// TIA Portal V19 export
FUNCTION "CollectAlarms" : Void   // FC61, LAD
TITLE = Alarm Collector Unit
// Collects alarms from the respective level and categorises the alarms into the different alarm classes. Filling the alarm DB with specific alarm messages which are defined in the comment of the defined alarm. The definition of possible alarms within a equipment is handled here.
// stored: Namespace Unit2.EM2, SetENOAutomatically false
   VAR_INPUT
      resetAlarms : Bool;
      disableAlarms : Bool;
   END_VAR
   VAR_OUTPUT
      commandsToUnit : "LUC_typeStateCommands";   // Feedback to the unit
   END_VAR
BEGIN

REGION Network 1: Reset Alarms
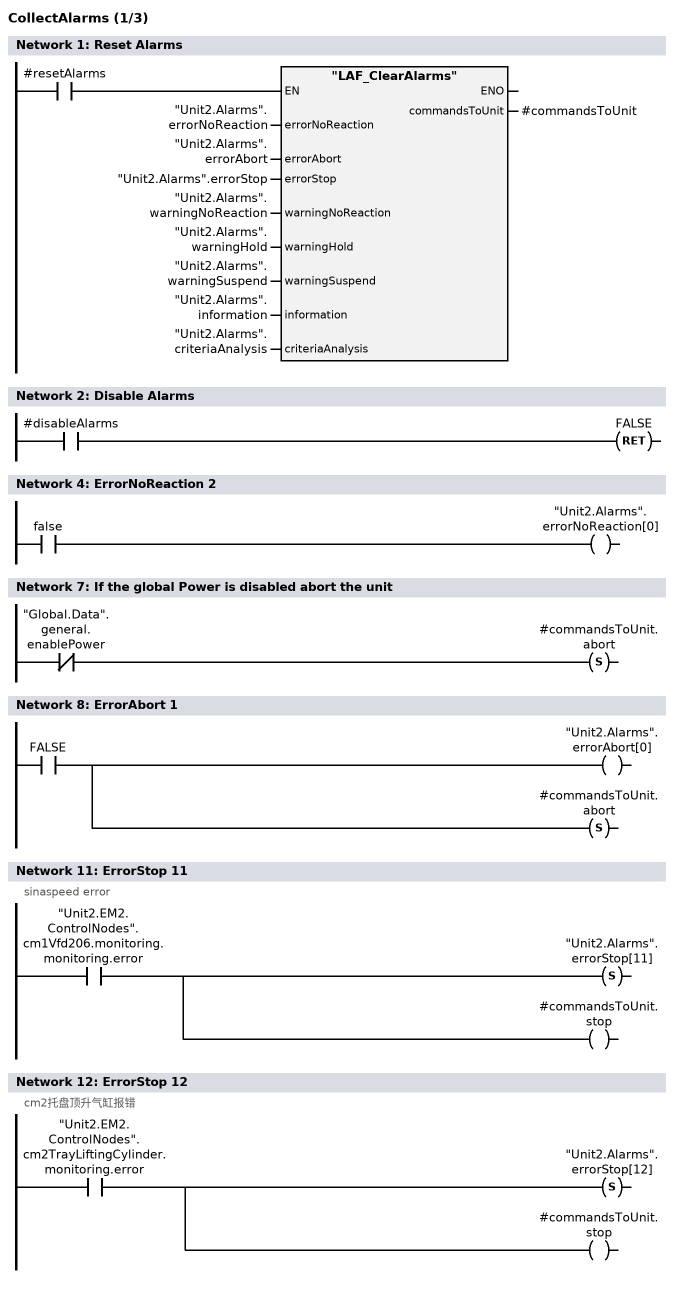
   RUNG wire#powerrail
      Contact( #resetAlarms )
      "LAF_ClearAlarms"(errorNoReaction := "Unit2.Alarms".errorNoReaction, errorAbort := "Unit2.Alarms".errorAbort, errorStop := "Unit2.Alarms".errorStop, warningNoReaction := "Unit2.Alarms".warningNoReaction, warningHold := "Unit2.Alarms".warningHold, warningSuspend := "Unit2.Alarms".warningSuspend, information := "Unit2.Alarms".information, criteriaAnalysis := "Unit2.Alarms".criteriaAnalysis, commandsToUnit => #commandsToUnit)
   END_RUNG
   // the same network as SCL:
   IF #resetAlarms THEN
       "LAF_ClearAlarms"(errorNoReaction := "Unit2.Alarms".errorNoReaction,
                         errorAbort := "Unit2.Alarms".errorAbort,
                         errorStop := "Unit2.Alarms".errorStop,
                         warningNoReaction := "Unit2.Alarms".warningNoReaction,
                         warningHold := "Unit2.Alarms".warningHold,
                         warningSuspend := "Unit2.Alarms".warningSuspend,
                         information := "Unit2.Alarms".information,
                         criteriaAnalysis := "Unit2.Alarms".criteriaAnalysis,
                         commandsToUnit => #commandsToUnit);
   END_IF;
END_REGION

REGION Network 2: Disable Alarms
   RUNG wire#powerrail
      Contact( #disableAlarms )
      ReturnCoil( FALSE )
   END_RUNG
   // the same network as SCL:
   IF #disableAlarms THEN
       ENO := FALSE;
       RETURN;
   END_IF;
END_REGION

REGION Network 3: *************** Error No Reaction ************************
END_REGION

REGION Network 4: ErrorNoReaction 2
   RUNG wire#powerrail
      Contact( false )
      Coil( "Unit2.Alarms".errorNoReaction[0] )
   END_RUNG
   // the same network as SCL:
   "Unit2.Alarms".errorNoReaction[0] := false;
END_REGION

REGION Network 6: *************** Error and Abort **************************
END_REGION

REGION Network 7: If the global Power is disabled abort the unit
   RUNG wire#powerrail
      I_Contact( "Global.Data".general.enablePower )
      S_Coil( #commandsToUnit.abort )
   END_RUNG
   // the same network as SCL:
   IF NOT "Global.Data".general.enablePower THEN #commandsToUnit.abort := TRUE; END_IF;
END_REGION

REGION Network 8: ErrorAbort 1
   RUNG wire#powerrail
      Contact( FALSE )
      wire#w1
      Coil( "Unit2.Alarms".errorAbort[0] )
   END_RUNG
   RUNG wire#w1
      S_Coil( #commandsToUnit.abort )
   END_RUNG
   // the same network as SCL:
   "Unit2.Alarms".errorAbort[0] := FALSE;
   IF FALSE THEN #commandsToUnit.abort := TRUE; END_IF;
END_REGION

REGION Network 10: *************** Error and Stop ***************************
END_REGION

REGION Network 11: ErrorStop 11
   // sinaspeed error
   RUNG wire#powerrail
      Contact( "Unit2.EM2.ControlNodes".cm1Vfd206.monitoring.monitoring.error )
      wire#w1
      S_Coil( "Unit2.Alarms".errorStop[11] )
   END_RUNG
   RUNG wire#w1
      Coil( #commandsToUnit.stop )
   END_RUNG
   // the same network as SCL:
   IF "Unit2.EM2.ControlNodes".cm1Vfd206.monitoring.monitoring.error THEN
       "Unit2.Alarms".errorStop[11] := TRUE;
   END_IF;
   #commandsToUnit.stop := "Unit2.EM2.ControlNodes".cm1Vfd206.monitoring.monitoring.error;
END_REGION

REGION Network 12: ErrorStop 12
   // cm2托盘顶升气缸报错
   RUNG wire#powerrail
      Contact( "Unit2.EM2.ControlNodes".cm2TrayLiftingCylinder.monitoring.error )
      wire#w1
      S_Coil( "Unit2.Alarms".errorStop[12] )
   END_RUNG
   RUNG wire#w1
      Coil( #commandsToUnit.stop )
   END_RUNG
   // the same network as SCL:
   IF "Unit2.EM2.ControlNodes".cm2TrayLiftingCylinder.monitoring.error THEN
       "Unit2.Alarms".errorStop[12] := TRUE;
   END_IF;
   #commandsToUnit.stop := "Unit2.EM2.ControlNodes".cm2TrayLiftingCylinder.monitoring.error;
END_REGION

REGION Network 13: ErrorStop 13
   // cm3电芯顶升气缸报错
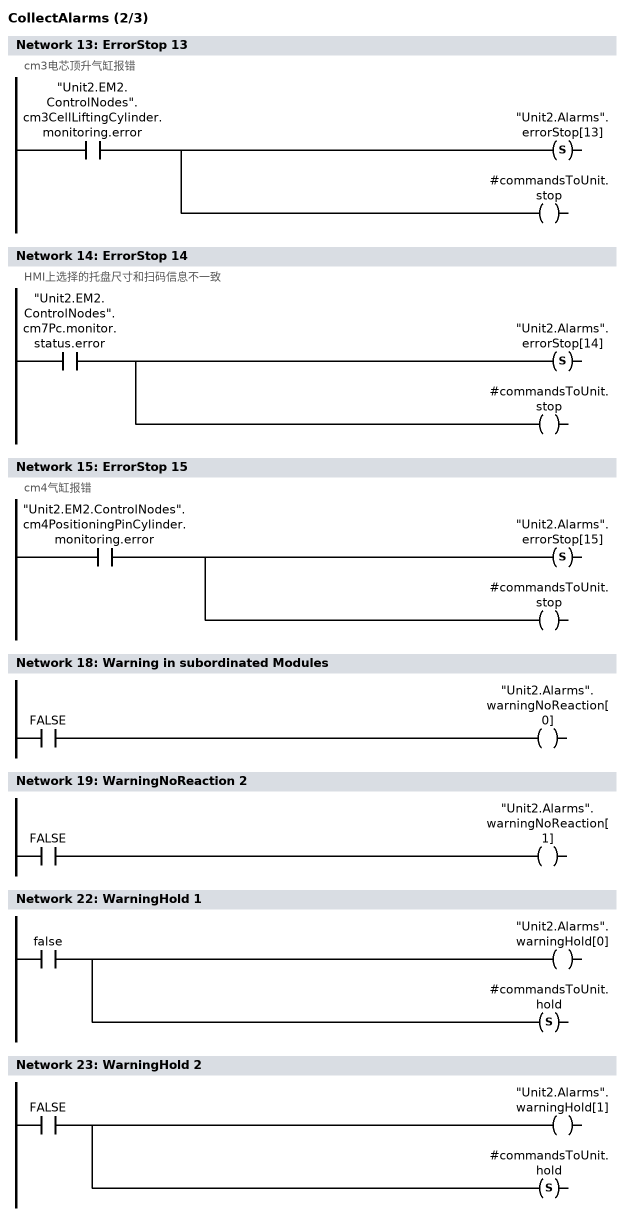
   RUNG wire#powerrail
      Contact( "Unit2.EM2.ControlNodes".cm3CellLiftingCylinder.monitoring.error )
      wire#w1
      S_Coil( "Unit2.Alarms".errorStop[13] )
   END_RUNG
   RUNG wire#w1
      Coil( #commandsToUnit.stop )
   END_RUNG
   // the same network as SCL:
   IF "Unit2.EM2.ControlNodes".cm3CellLiftingCylinder.monitoring.error THEN
       "Unit2.Alarms".errorStop[13] := TRUE;
   END_IF;
   #commandsToUnit.stop := "Unit2.EM2.ControlNodes".cm3CellLiftingCylinder.monitoring.error;
END_REGION

REGION Network 14: ErrorStop 14
   // HMI上选择的托盘尺寸和扫码信息不一致
   RUNG wire#powerrail
      Contact( "Unit2.EM2.ControlNodes".cm7Pc.monitor.status.error )
      wire#w1
      S_Coil( "Unit2.Alarms".errorStop[14] )
   END_RUNG
   RUNG wire#w1
      Coil( #commandsToUnit.stop )
   END_RUNG
   // the same network as SCL:
   IF "Unit2.EM2.ControlNodes".cm7Pc.monitor.status.error THEN "Unit2.Alarms".errorStop[14] := TRUE; END_IF;
   #commandsToUnit.stop := "Unit2.EM2.ControlNodes".cm7Pc.monitor.status.error;
END_REGION

REGION Network 15: ErrorStop 15
   // cm4气缸报错
   RUNG wire#powerrail
      Contact( "Unit2.EM2.ControlNodes".cm4PositioningPinCylinder.monitoring.error )
      wire#w1
      S_Coil( "Unit2.Alarms".errorStop[15] )
   END_RUNG
   RUNG wire#w1
      Coil( #commandsToUnit.stop )
   END_RUNG
   // the same network as SCL:
   IF "Unit2.EM2.ControlNodes".cm4PositioningPinCylinder.monitoring.error THEN
       "Unit2.Alarms".errorStop[15] := TRUE;
   END_IF;
   #commandsToUnit.stop := "Unit2.EM2.ControlNodes".cm4PositioningPinCylinder.monitoring.error;
END_REGION

REGION Network 17: *************** Warning No Reaction **********************
END_REGION

REGION Network 18: Warning in subordinated Modules
   RUNG wire#powerrail
      Contact( FALSE )
      Coil( "Unit2.Alarms".warningNoReaction[0] )
   END_RUNG
   // the same network as SCL:
   "Unit2.Alarms".warningNoReaction[0] := FALSE;
END_REGION

REGION Network 19: WarningNoReaction 2
   RUNG wire#powerrail
      Contact( FALSE )
      Coil( "Unit2.Alarms".warningNoReaction[1] )
   END_RUNG
   // the same network as SCL:
   "Unit2.Alarms".warningNoReaction[1] := FALSE;
END_REGION

REGION Network 21: *************** Warning Hold **************************
END_REGION

REGION Network 22: WarningHold 1
   RUNG wire#powerrail
      Contact( false )
      wire#w1
      Coil( "Unit2.Alarms".warningHold[0] )
   END_RUNG
   RUNG wire#w1
      S_Coil( #commandsToUnit.hold )
   END_RUNG
   // the same network as SCL:
   "Unit2.Alarms".warningHold[0] := false;
   IF false THEN #commandsToUnit.hold := TRUE; END_IF;
END_REGION

REGION Network 23: WarningHold 2
   RUNG wire#powerrail
      Contact( FALSE )
      wire#w1
      Coil( "Unit2.Alarms".warningHold[1] )
   END_RUNG
   RUNG wire#w1
      S_Coil( #commandsToUnit.hold )
   END_RUNG
   // the same network as SCL:
   "Unit2.Alarms".warningHold[1] := FALSE;
   IF FALSE THEN #commandsToUnit.hold := TRUE; END_IF;
END_REGION

REGION Network 25: *************** Warning Suspend ***********************
END_REGION

REGION Network 26: WarningSuspend 1
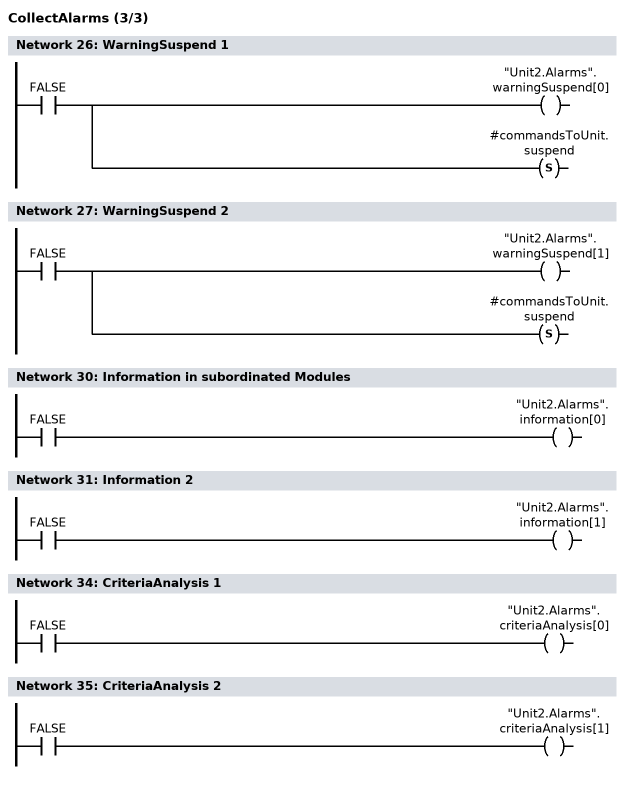
   RUNG wire#powerrail
      Contact( FALSE )
      wire#w1
      Coil( "Unit2.Alarms".warningSuspend[0] )
   END_RUNG
   RUNG wire#w1
      S_Coil( #commandsToUnit.suspend )
   END_RUNG
   // the same network as SCL:
   "Unit2.Alarms".warningSuspend[0] := FALSE;
   IF FALSE THEN #commandsToUnit.suspend := TRUE; END_IF;
END_REGION

REGION Network 27: WarningSuspend 2
   RUNG wire#powerrail
      Contact( FALSE )
      wire#w1
      Coil( "Unit2.Alarms".warningSuspend[1] )
   END_RUNG
   RUNG wire#w1
      S_Coil( #commandsToUnit.suspend )
   END_RUNG
   // the same network as SCL:
   "Unit2.Alarms".warningSuspend[1] := FALSE;
   IF FALSE THEN #commandsToUnit.suspend := TRUE; END_IF;
END_REGION

REGION Network 29: *************** Information *****************************
END_REGION

REGION Network 30: Information in subordinated Modules
   RUNG wire#powerrail
      Contact( FALSE )
      Coil( "Unit2.Alarms".information[0] )
   END_RUNG
   // the same network as SCL:
   "Unit2.Alarms".information[0] := FALSE;
END_REGION

REGION Network 31: Information 2
   RUNG wire#powerrail
      Contact( FALSE )
      Coil( "Unit2.Alarms".information[1] )
   END_RUNG
   // the same network as SCL:
   "Unit2.Alarms".information[1] := FALSE;
END_REGION

REGION Network 33: *************** CriteriaAnalysis **************************
END_REGION

REGION Network 34: CriteriaAnalysis 1
   RUNG wire#powerrail
      Contact( FALSE )
      Coil( "Unit2.Alarms".criteriaAnalysis[0] )
   END_RUNG
   // the same network as SCL:
   "Unit2.Alarms".criteriaAnalysis[0] := FALSE;
END_REGION

REGION Network 35: CriteriaAnalysis 2
   RUNG wire#powerrail
      Contact( FALSE )
      Coil( "Unit2.Alarms".criteriaAnalysis[1] )
   END_RUNG
   // the same network as SCL:
   "Unit2.Alarms".criteriaAnalysis[1] := FALSE;
END_REGION
END_FUNCTION
